{attribute 'GeneratedUsingTerminal: EJ1918-0000-0017'}
{attribute addProperty BoxType "EJ1918-0000-0017"}
{attribute addProperty Id "FSOEAT %I*FSOE_9F04885D17"}
{attribute addProperty CRC "3328292746"}
{attribute addProperty Size "17"}
TYPE FSoE_Inputs_C661B78A EXTENDS InputBase_8311D824 :
STRUCT
	{attribute addProperty Name "FSOE"}
	FSOE AT %I* : FSOE_9F04885D;
END_STRUCT
END_TYPE

(* stored: Version 1.2.0.0, ProductVersion 3.1.4024.9
   DUT FSoE_Inputs_C661B78A: Id {350bbccf-6d03-4aac-8dfe-9c9dc091ceef} *)
